{attribute addProperty BoxType "EK1100-0000-0018"}
{attribute addProperty Id "Beckhoff_EM2xxxEK1122Beckhoff_EM2xxxEK1122_264CF75A162A_0001_EM2042_0000_0016EM2042_5A2A5F2915219A_0002_EM2042_0000_0017EM2042_5A2A5F2915219"}
{attribute addProperty CRC "693890983"}
{attribute addProperty SizeInBites "320"}
{attribute addProperty SizeInBytes "40"}
TYPE Beckhoff_EM2xxx_295BEFA7 EXTENDS EK1100_179A0949 :
STRUCT
	{attribute addProperty Name "Beckhoff_EM2xxxEK1122"}
	Beckhoff_EM2xxxEK1122 : Beckhoff_EM2xxxEK1122_264CF75A;
	{attribute addProperty Name "A_0001_EM2042_0000_0016"}
	A_0001_EM2042_0000_0016 : EM2042_5A2A5F29;
	{attribute addProperty Name "A_0002_EM2042_0000_0017"}
	A_0002_EM2042_0000_0017 : EM2042_5A2A5F29;
END_STRUCT
END_TYPE

(* stored: Version 1.2.0.0, ProductVersion 3.1.4024.9
   DUT Beckhoff_EM2xxx_295BEFA7: Id {2daf9406-9786-4e21-8c60-06daace9c32f} *)
